// SIMATIC S7-200 project (STEP 7-Micro/WIN), CPU 224XP CN REL 02.01

SYMBOL_TABLE USER1
Enc_A            I0.0     // Encoder Fase A
Enc_B            I0.1     // Encoder Fase B
Enc_C            I0.2     // Encoder Fase C (Indice)
Sens_Objeto      I0.3     // Sensor deteccion de pieza en entrada
Sens_Fibra       I0.4     // Sensor fibra Omron (Clasificacion)
Sens_Mag         I0.5     // Sensor magnetico (Clasificacion)
Extendido_C1     I0.7     // Confirmacion extension cilindro rampa 1
Extendido_C2     I1.0     // Confirmacion extension cilindro rampa 2
Extendido_C3     I1.1     // Confirmacion extension cilindro rampa 3
Btn_Paro         I1.2     // Pulsador rojo de paro
Btn_Marcha       I1.3     // Pulsador verde de marcha
Seta_Emerg       I1.4     // Zeta de emergencia (NC)
Selector         I1.5     // Selector rotatorio de modo
Motor_Cinta      Q0.0     // Mando marcha variador
Motor_Dir        Q0.1     // Mando de direccion del motor
V_Cil1           Q0.4     // Valvula cilindro rampa 1
V_Cil2           Q0.5     // Valvula cilindro rampa 2
V_Cil3           Q0.6     // Valvula cilindro rampa 3
Lamp_Amarilla    Q0.7     // Luz de advertencia
Lamp_Verde       Q1.0     // Luz de marcha
Lamp_Roja        Q1.1     // Luz de paro o falla
Salida_Analog    AQW0     // Consigna velocidad variador (0-32000)
Pos_Real         VD100    // Posicion actual en cuentas (REAL)
Pos_Last         VD104    // Posicion ciclo anterior (REAL)
Vel_Actual       VD108    // Velocidad calculada en cuentas/s (REAL)
Setpoint         VD112    // Posicion objetivo para el controlador (REAL)
Accion_Ctrl      VD116    // U calculada por realimentacion estados (REAL)
K1               VD120    // Ganancia de posicion (REAL)
K2               VD124    // Ganancia de velocidad (REAL)
N                VD132    // Ganancia de pre-compensacion (REAL)
U_Abs            VD128    // Magnitud absoluta de accion de control (REAL)
Coord_Rampa      VD300    // Coordenada de rampa seleccionada (REAL)
P0_Reposo        M0.0     // Estado de espera inicial
P1_Avanzar       M0.1     // Movimiento hacia zona de sensores
P2_Ident         M0.2     // Clasificacion al vuelo (Posicion 500)
P3_Viaje         M0.3     // Movimiento hacia rampa objetivo
P4_Expulsar      M0.4     // Activacion de cilindro empujador
P5_Final         M0.5     // Retorno de actuadores y reset
T0_Inicio        M1.0     // Disparo: Marcha + Pieza
T1_Pos500        M1.1     // Disparo: Llegada a cuenta 500
T2_Clasificado   M1.2     // Disparo: Carga de coordenada terminada
T3_Target        M1.3     // Disparo: Llegada a rampa objetivo
T4_Push_OK       M1.4     // Disparo: Expulsion confirmada
T5_Fin_Ciclo     M1.5     // Disparo: Sistema restaurado
Ev_Marcha        M2.0     // Evento: Orden de inicio y Seta OK
Ev_Pieza_In      M2.1     // Evento: Pieza detectada en entrada
Ev_P500          M2.2     // Evento: Encoder >= 500
Ev_PRampa        M2.3     // Evento: Encoder >= Coordenada Rampa
Ev_Cil_Ext       M2.4     // Evento: Uno de los cilindros extendido
Ack_MS           V0.1     // Reconocimiento marcha Unidad de Seleccion
Marcha_S         V1.1     // Solicitud de marcha para la Unidad de Seleccion
Sel_OK           V0.2     // Unidad de Seleccion disponible
Pieza_Metal      V0.3     // Indica si la pieza atendida es totalmente metalica
Pieza_Mixta      V0.4     // Indica si la pieza atendida es mixta (metal-plastico o plastico-metal)
Pieza_Plastica   V0.5     // Indica si la pieza atendida es totalemnte plastica
END_SYMBOL_TABLE

SYMBOL_TABLE S7-200 Symbols
Always_On        SM0.0    // 始终接通为 ON
First_Scan_On    SM0.1    // 仅第一个扫描周期中接通为 ON
Time_0_Intrvl    SMB34    // 定时中断 0 的时间间隔（从 1 至 255，以 1 毫秒为增量）。
HSC0_Ctrl        SMB37    // HSC0 设置与控制
HSC0_CV          SMD38    // HSC0 的新当前值
HSC0_PV          SMD42    // HSC0 的新预置值
END_SYMBOL_TABLE

ORGANIZATION_BLOCK MAIN:OB1
TITLE=UNIDAD DE SELECCION - RED DE PETRI + CONTROL DE ESTADOS
//  MODULO 1: INICIALIZACION
//  MODULO 2: EVENTOS
//  MODULO 3: DISPARO
//  MODULO 4: DINAMICA
//  MODULO 5: ACCIONES
//  MODULO 1: INICIALIZACION
BEGIN
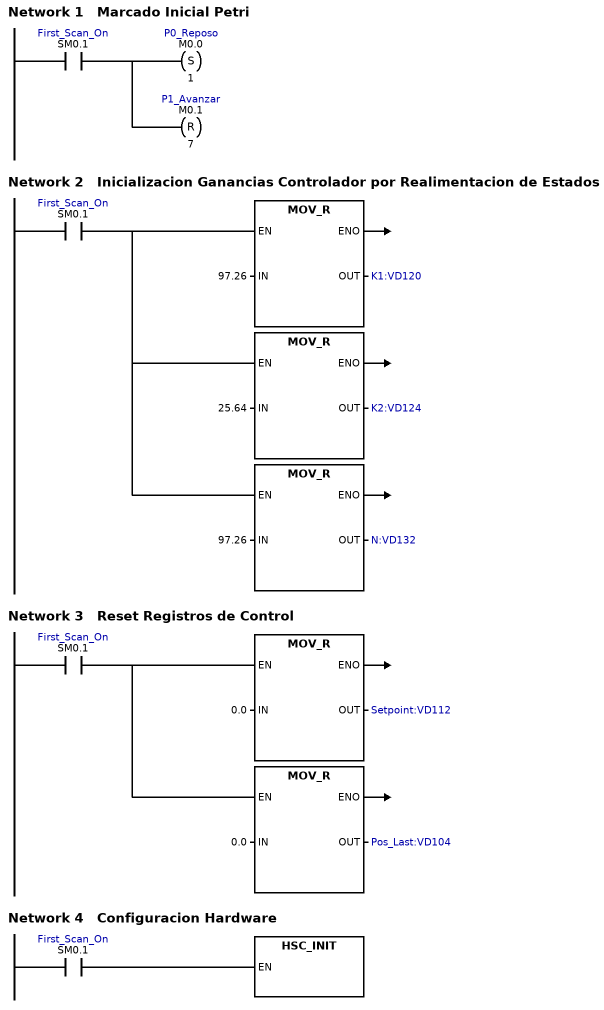
Network 1 //  Marcado Inicial Petri
// P0 Reposo activo
// Limpiar marcas P1 a M0.7
LD     First_Scan_On:SM0.1
S      P0_Reposo:M0.0, 1
R      P1_Avanzar:M0.1, 7
Network 2 //  Inicializacion Ganancias Controlador por Realimentacion de Estados
// K1
// K2
// N
LD     First_Scan_On:SM0.1
MOVR   97.26, K1:VD120
MOVR   25.64, K2:VD124
MOVR   97.26, N:VD132
Network 3 //  Reset Registros de Control
// Setpoint Inicial
// Reset Pos_Last
LD     First_Scan_On:SM0.1
MOVR   0.0, Setpoint:VD112
MOVR   0.0, Pos_Last:VD104
Network 4 //  Configuracion Hardware
// Inicializar HSC0
LD     First_Scan_On:SM0.1
CALL   HSC_INIT:SBR1
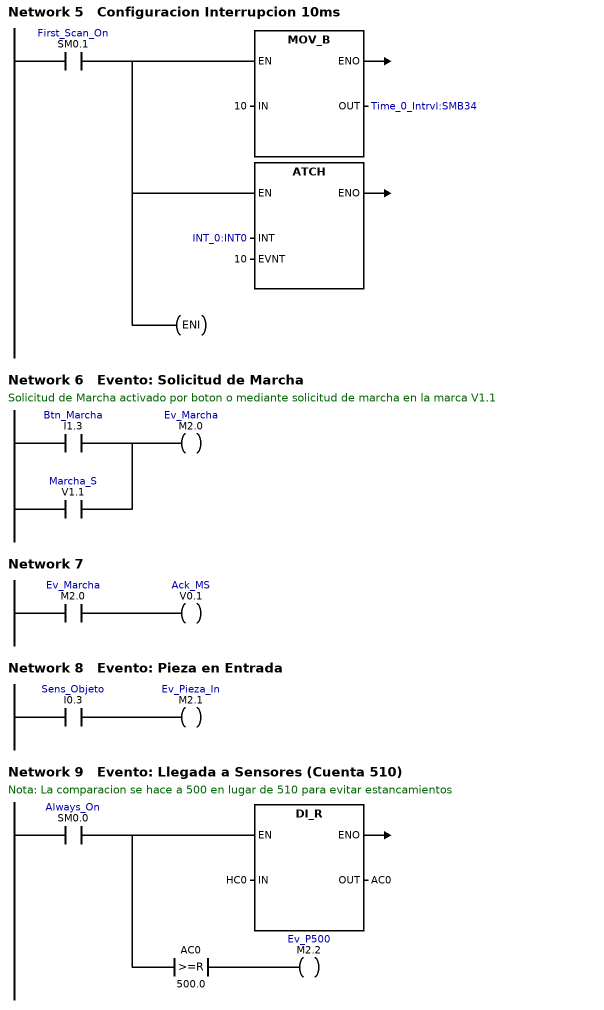
Network 5 //  Configuracion Interrupcion 10ms
// MODULO 2: EVENTOS (CAPTURA DE SENSORES Y COMPARADORES)
LD     First_Scan_On:SM0.1
MOVB   10, Time_0_Intrvl:SMB34
ATCH   INT_0:INT0, 10
ENI
Network 6 //  Evento: Solicitud de Marcha
//  Solicitud de Marcha activado por boton o mediante solicitud de marcha en la marca V1.1
LD     Btn_Marcha:I1.3
O      Marcha_S:V1.1
=      Ev_Marcha:M2.0
Network 7
LD     Ev_Marcha:M2.0
=      Ack_MS:V0.1
Network 8 //  Evento: Pieza en Entrada
LD     Sens_Objeto:I0.3
=      Ev_Pieza_In:M2.1
Network 9 //  Evento: Llegada a Sensores (Cuenta 510)
// Nota: La comparacion se hace a 500 en lugar de 510 para evitar estancamientos
LD     Always_On:SM0.0
DTR    HC0, AC0
AR>=   AC0, 500.0
=      Ev_P500:M2.2
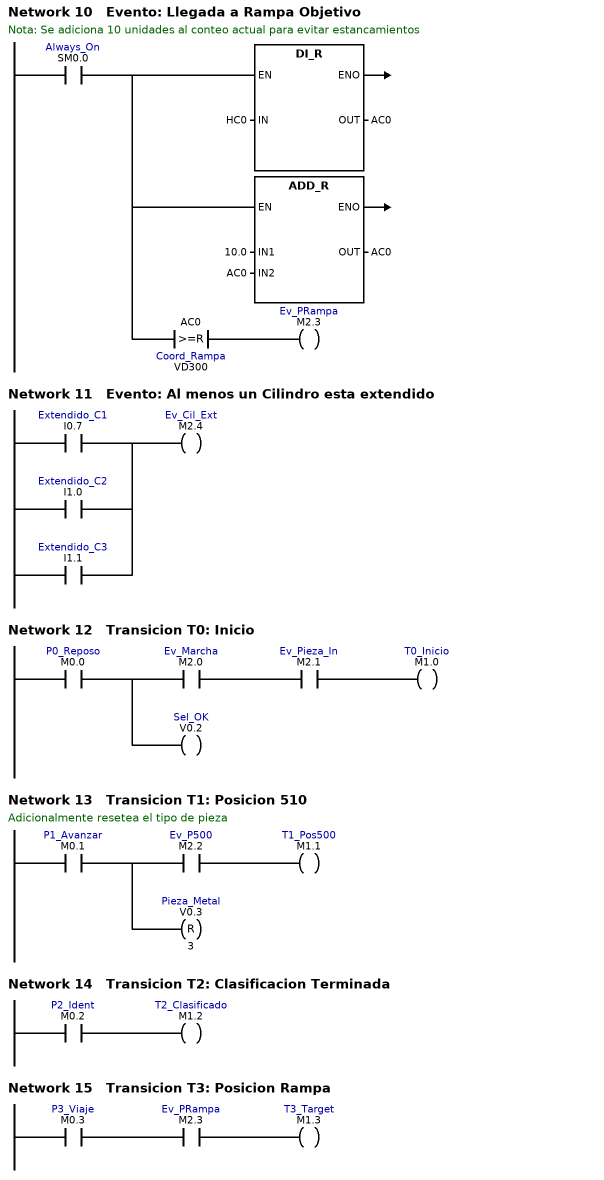
Network 10 //  Evento: Llegada a Rampa Objetivo
// Nota: Se adiciona 10 unidades al conteo actual para evitar estancamientos
LD     Always_On:SM0.0
DTR    HC0, AC0
+R     10.0, AC0
AR>=   AC0, Coord_Rampa:VD300
=      Ev_PRampa:M2.3
Network 11 //  Evento: Al menos un Cilindro esta extendido
// MODULO 3: CONDICIONES DE DISPARO (FIRING)
LD     Extendido_C1:I0.7
O      Extendido_C2:I1.0
O      Extendido_C3:I1.1
=      Ev_Cil_Ext:M2.4
Network 12 //  Transicion T0: Inicio
LD     P0_Reposo:M0.0
LPS
A      Ev_Marcha:M2.0
A      Ev_Pieza_In:M2.1
=      T0_Inicio:M1.0
LPP
=      Sel_OK:V0.2
Network 13 //  Transicion T1: Posicion 510
// Adicionalmente resetea el tipo de pieza
LD     P1_Avanzar:M0.1
LPS
A      Ev_P500:M2.2
=      T1_Pos500:M1.1
LPP
R      Pieza_Metal:V0.3, 3
Network 14 //  Transicion T2: Clasificacion Terminada
LD     P2_Ident:M0.2
=      T2_Clasificado:M1.2
Network 15 //  Transicion T3: Posicion Rampa
LD     P3_Viaje:M0.3
A      Ev_PRampa:M2.3
=      T3_Target:M1.3
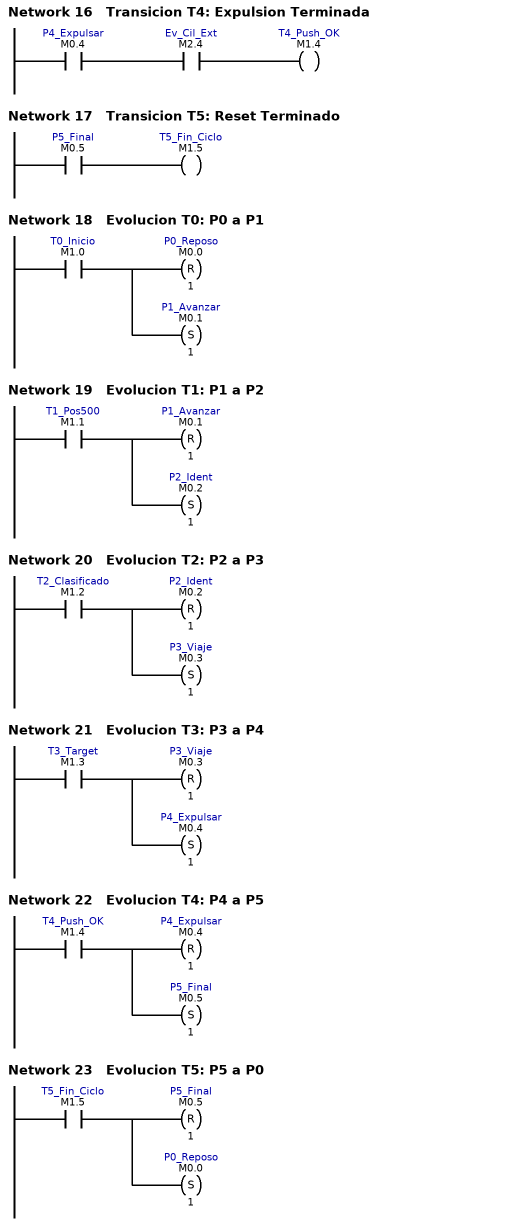
Network 16 //  Transicion T4: Expulsion Terminada
LD     P4_Expulsar:M0.4
A      Ev_Cil_Ext:M2.4
=      T4_Push_OK:M1.4
Network 17 //  Transicion T5: Reset Terminado
// MODULO 4: DINAMICA DE LA RED (EVOLUCION)
LD     P5_Final:M0.5
=      T5_Fin_Ciclo:M1.5
Network 18 //  Evolucion T0: P0 a P1
LD     T0_Inicio:M1.0
R      P0_Reposo:M0.0, 1
S      P1_Avanzar:M0.1, 1
Network 19 //  Evolucion T1: P1 a P2
LD     T1_Pos500:M1.1
R      P1_Avanzar:M0.1, 1
S      P2_Ident:M0.2, 1
Network 20 //  Evolucion T2: P2 a P3
LD     T2_Clasificado:M1.2
R      P2_Ident:M0.2, 1
S      P3_Viaje:M0.3, 1
Network 21 //  Evolucion T3: P3 a P4
LD     T3_Target:M1.3
R      P3_Viaje:M0.3, 1
S      P4_Expulsar:M0.4, 1
Network 22 //  Evolucion T4: P4 a P5
LD     T4_Push_OK:M1.4
R      P4_Expulsar:M0.4, 1
S      P5_Final:M0.5, 1
Network 23 //  Evolucion T5: P5 a P0
LD     T5_Fin_Ciclo:M1.5
R      P5_Final:M0.5, 1
S      P0_Reposo:M0.0, 1
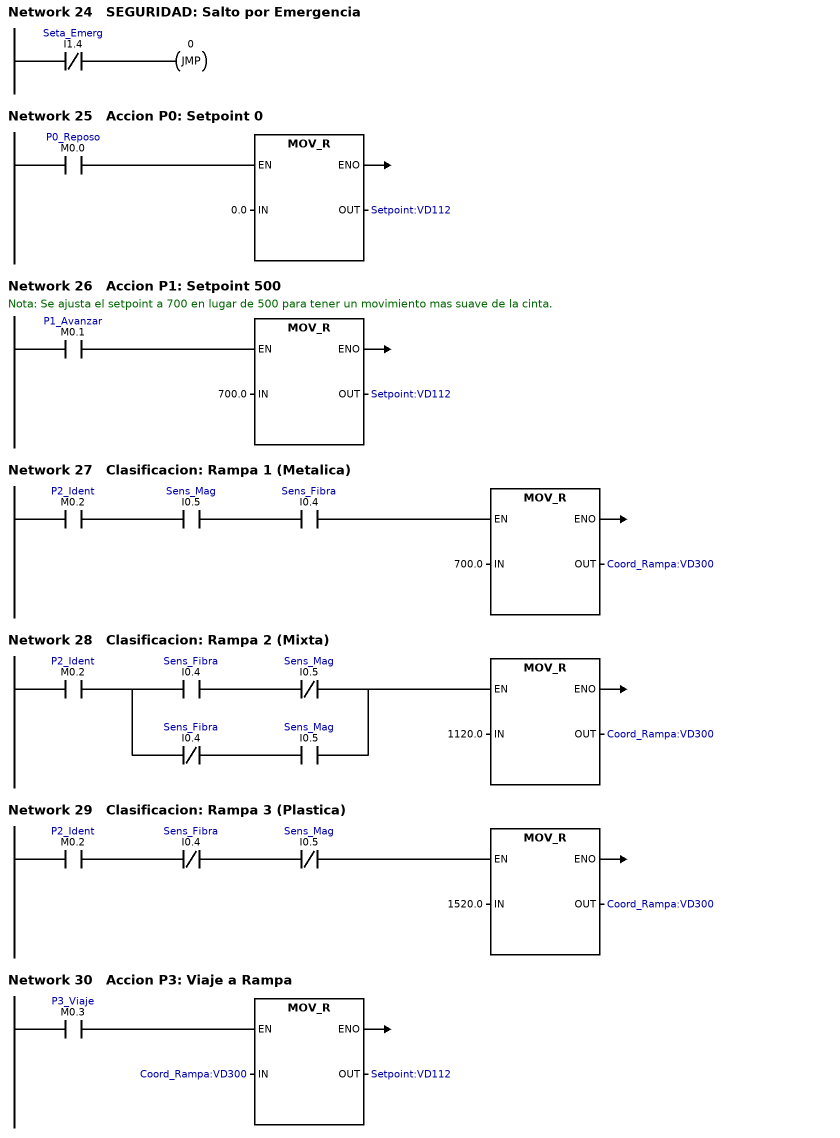
Network 24 //  SEGURIDAD: Salto por Emergencia
// MODULO 5: ACCIONES (SALIDAS Y SETPOINTS)
LDN    Seta_Emerg:I1.4
JMP    0
Network 25 //  Accion P0: Setpoint 0
LD     P0_Reposo:M0.0
MOVR   0.0, Setpoint:VD112
Network 26 //  Accion P1: Setpoint 500
// Nota: Se ajusta el setpoint a 700 en lugar de 500 para tener un movimiento mas suave de la cinta.
LD     P1_Avanzar:M0.1
MOVR   700.0, Setpoint:VD112
Network 27 //  Clasificacion: Rampa 1 (Metalica)
LD     P2_Ident:M0.2
A      Sens_Mag:I0.5
A      Sens_Fibra:I0.4
MOVR   700.0, Coord_Rampa:VD300
Network 28 //  Clasificacion: Rampa 2 (Mixta)
LD     P2_Ident:M0.2
LD     Sens_Fibra:I0.4
AN     Sens_Mag:I0.5
LDN    Sens_Fibra:I0.4
A      Sens_Mag:I0.5
OLD
ALD
MOVR   1120.0, Coord_Rampa:VD300
Network 29 //  Clasificacion: Rampa 3 (Plastica)
LD     P2_Ident:M0.2
AN     Sens_Fibra:I0.4
AN     Sens_Mag:I0.5
MOVR   1520.0, Coord_Rampa:VD300
Network 30 //  Accion P3: Viaje a Rampa
LD     P3_Viaje:M0.3
MOVR   Coord_Rampa:VD300, Setpoint:VD112
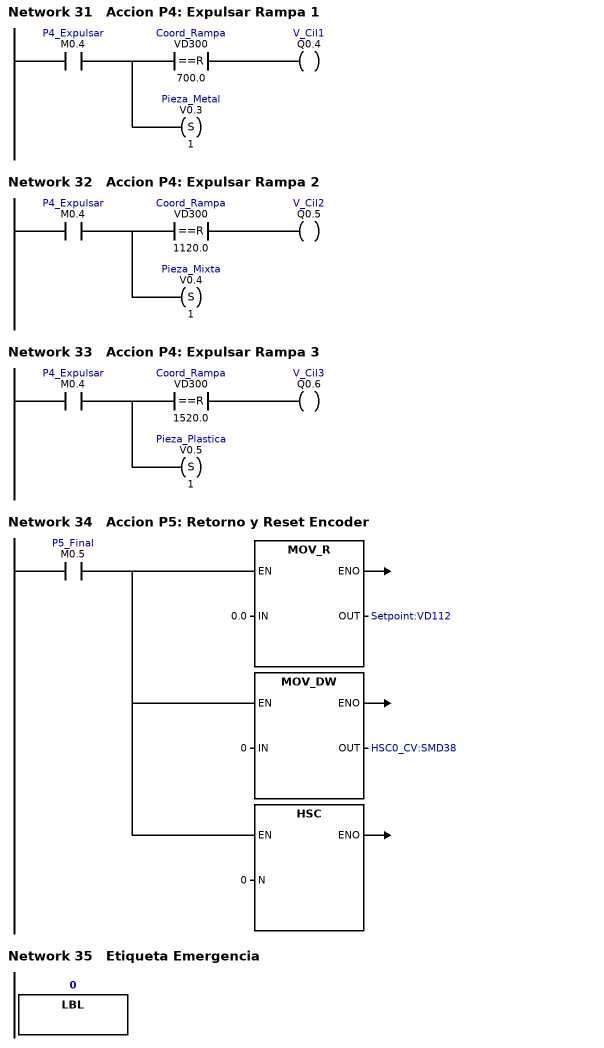
Network 31 //  Accion P4: Expulsar Rampa 1
LD     P4_Expulsar:M0.4
LPS
AR=    Coord_Rampa:VD300, 700.0
=      V_Cil1:Q0.4
LPP
S      Pieza_Metal:V0.3, 1
Network 32 //  Accion P4: Expulsar Rampa 2
LD     P4_Expulsar:M0.4
LPS
AR=    Coord_Rampa:VD300, 1120.0
=      V_Cil2:Q0.5
LPP
S      Pieza_Mixta:V0.4, 1
Network 33 //  Accion P4: Expulsar Rampa 3
LD     P4_Expulsar:M0.4
LPS
AR=    Coord_Rampa:VD300, 1520.0
=      V_Cil3:Q0.6
LPP
S      Pieza_Plastica:V0.5, 1
Network 34 //  Accion P5: Retorno y Reset Encoder
LD     P5_Final:M0.5
MOVR   0.0, Setpoint:VD112
MOVD   0, HSC0_CV:SMD38
HSC    0
Network 35 //  Etiqueta Emergencia
LBL    0
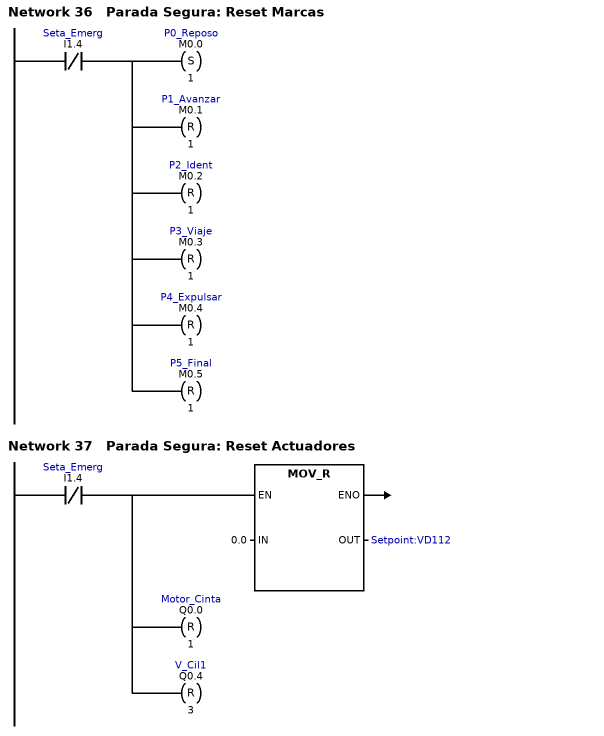
Network 36 //  Parada Segura: Reset Marcas
LDN    Seta_Emerg:I1.4
S      P0_Reposo:M0.0, 1
R      P1_Avanzar:M0.1, 1
R      P2_Ident:M0.2, 1
R      P3_Viaje:M0.3, 1
R      P4_Expulsar:M0.4, 1
R      P5_Final:M0.5, 1
Network 37 //  Parada Segura: Reset Actuadores
LDN    Seta_Emerg:I1.4
MOVR   0.0, Setpoint:VD112
R      Motor_Cinta:Q0.0, 1
R      V_Cil1:Q0.4, 3
END_ORGANIZATION_BLOCK

SUBROUTINE_BLOCK HSC_INIT:SBR1
TITLE=INICIALIZACION ENCODER HSC0
BEGIN
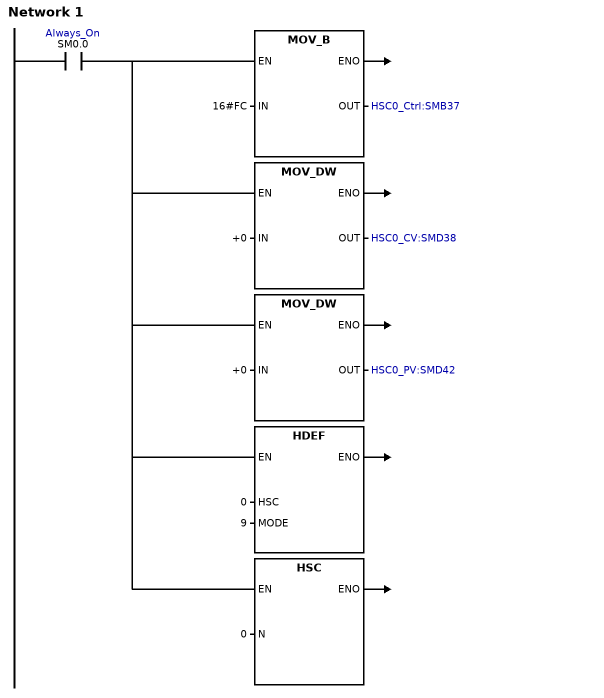
Network 1
LD     Always_On:SM0.0
MOVB   16#FC, HSC0_Ctrl:SMB37
MOVD   +0, HSC0_CV:SMD38
MOVD   +0, HSC0_PV:SMD42
HDEF   0, 9
HSC    0
END_SUBROUTINE_BLOCK

INTERRUPT_BLOCK INT_0:INT0
TITLE=CONTROLADOR REALIMENTACION ESTADOS 10ms
BEGIN
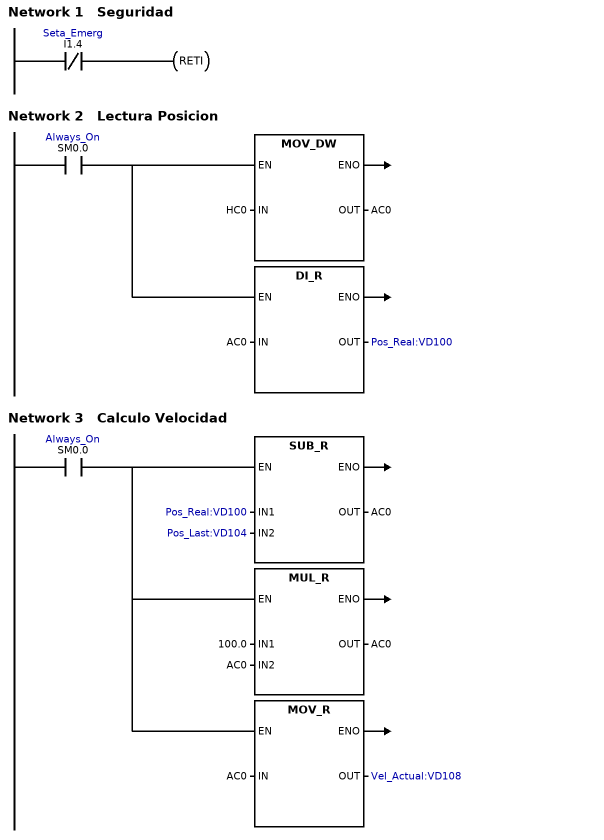
Network 1 //  Seguridad
LDN    Seta_Emerg:I1.4
CRETI
Network 2 //  Lectura Posicion
LD     Always_On:SM0.0
MOVD   HC0, AC0
DTR    AC0, Pos_Real:VD100
Network 3 //  Calculo Velocidad
LD     Always_On:SM0.0
MOVR   Pos_Real:VD100, AC0
-R     Pos_Last:VD104, AC0
*R     100.0, AC0
MOVR   AC0, Vel_Actual:VD108
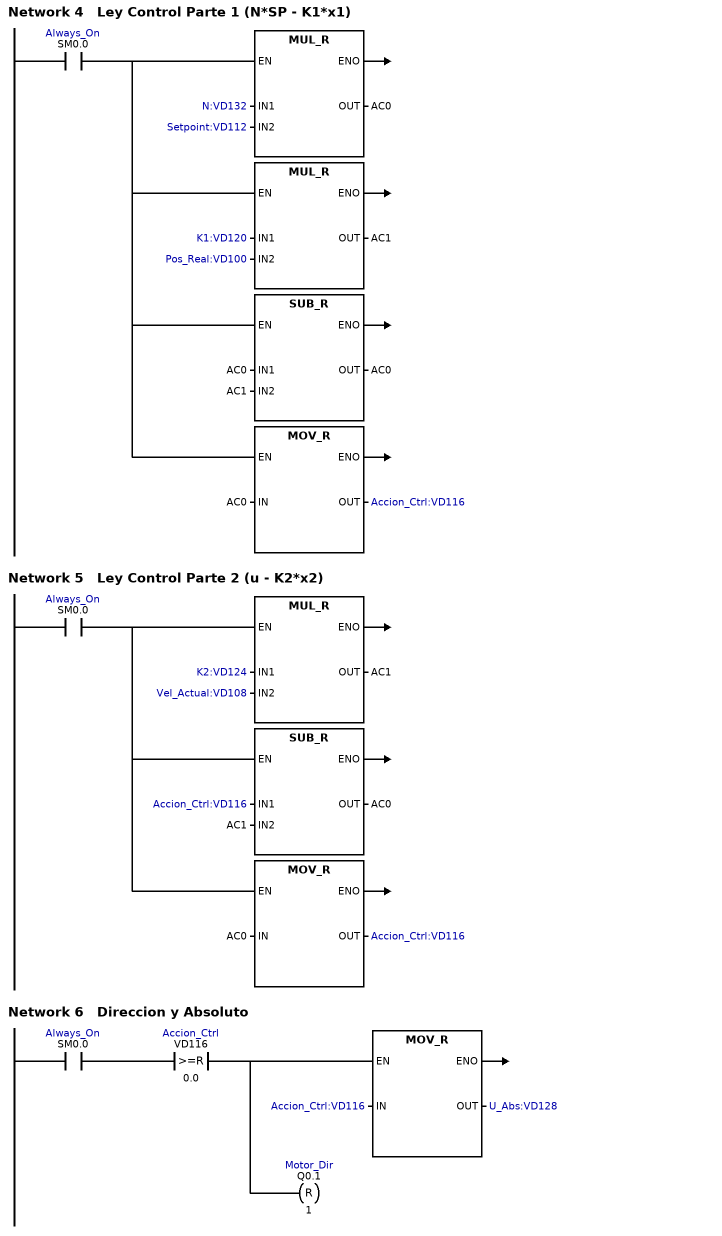
Network 4 //  Ley Control Parte 1 (N*SP - K1*x1)
LD     Always_On:SM0.0
MOVR   N:VD132, AC0
*R     Setpoint:VD112, AC0
MOVR   K1:VD120, AC1
*R     Pos_Real:VD100, AC1
-R     AC1, AC0
MOVR   AC0, Accion_Ctrl:VD116
Network 5 //  Ley Control Parte 2 (u - K2*x2)
LD     Always_On:SM0.0
MOVR   K2:VD124, AC1
*R     Vel_Actual:VD108, AC1
MOVR   Accion_Ctrl:VD116, AC0
-R     AC1, AC0
MOVR   AC0, Accion_Ctrl:VD116
Network 6 //  Direccion y Absoluto
LD     Always_On:SM0.0
AR>=   Accion_Ctrl:VD116, 0.0
MOVR   Accion_Ctrl:VD116, U_Abs:VD128
R      Motor_Dir:Q0.1, 1
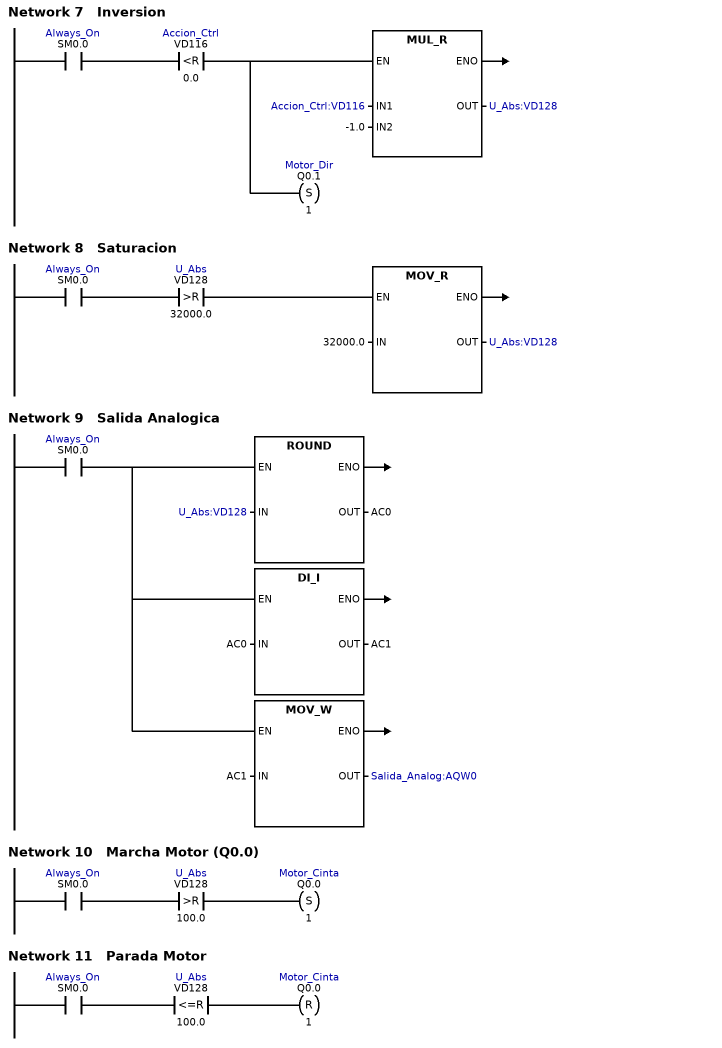
Network 7 //  Inversion
LD     Always_On:SM0.0
AR<    Accion_Ctrl:VD116, 0.0
MOVR   Accion_Ctrl:VD116, U_Abs:VD128
*R     -1.0, U_Abs:VD128
S      Motor_Dir:Q0.1, 1
Network 8 //  Saturacion
LD     Always_On:SM0.0
AR>    U_Abs:VD128, 32000.0
MOVR   32000.0, U_Abs:VD128
Network 9 //  Salida Analogica
LD     Always_On:SM0.0
ROUND  U_Abs:VD128, AC0
DTI    AC0, AC1
MOVW   AC1, Salida_Analog:AQW0
Network 10 //  Marcha Motor (Q0.0)
LD     Always_On:SM0.0
AR>    U_Abs:VD128, 100.0
S      Motor_Cinta:Q0.0, 1
Network 11 //  Parada Motor
LD     Always_On:SM0.0
AR<=   U_Abs:VD128, 100.0
R      Motor_Cinta:Q0.0, 1
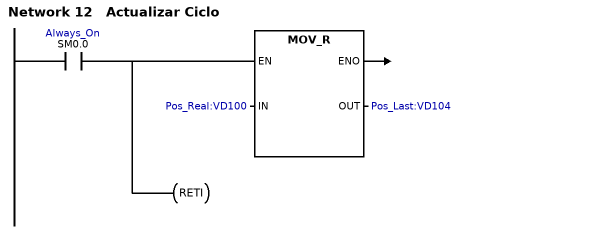
Network 12 //  Actualizar Ciclo
LD     Always_On:SM0.0
MOVR   Pos_Real:VD100, Pos_Last:VD104
CRETI
END_INTERRUPT_BLOCK
